{attribute 'linkalways'} 
{attribute 'no_explicit_call' := 'This FB is a CLASS and must be accessed using methods or properties'}
{attribute 'enable_dynamic_creation'}
FUNCTION_BLOCK Node_F_VN_ElementwiseLog EXTENDS VisionNode
VAR
    ipSrcImage : _ITcVnImage;
    ipDestImage : _ITcVnImage;
    hrPrev : _HRESULT(S_OK);
	hresult : _HRESULT(S_OK);
END_VAR

METHOD PUBLIC  Clone : I_Node
VAR
	pNode : POINTER TO Node_F_VN_ElementwiseLog;
END_VAR
pNode := __NEW(Node_F_VN_ElementwiseLog);
Clone := pNode^;
END_METHOD

METHOD FB_init : BOOL
VAR_INPUT
	bInitRetains : BOOL; // if TRUE, the retain variables are initialized (warm start / cold start)
	bInCopyCode : BOOL;  // if TRUE, the instance afterwards gets moved into the copy code (online change)
END_VAR
AddInput('ipSrcImage', ipSrcImage);
AddInput('hrPrev', hrPrev);
AddOutput('ipDestImage', ipDestImage);
AddOutput('hresult',hresult);
END_METHOD

METHOD PROTECTED OnExecute : HRESULT
hresult.Value := F_VN_ElementwiseLog(
    ipSrcImage := ipSrcImage.Value,
	ipDestImage := ipDestImage.Value,
	hrPrev:= hrPrev.Value);
END_METHOD

METHOD PUBLIC PreExecutionCheck
VAR_INPUT
	Check : I_PreExecutionChecks;
END_VAR
IF FAILED(hrPrev.Value) THEN
    RETURN;
END_IF

Check.IsTrue(ipSrcImage.IsValid, 'ipSrcImage must contain an image');
Check.IsTrue((ipSrcImage.IsPixelDepth(32) OR
              ipSrcImage.IsPixelDepth(64)), 'ipSrcImage must have 32 or 64 bit pixel depth');
END_METHOD

END_FUNCTION_BLOCK

(* stored: Version 1.1.0.1, ProductVersion 3.1.4024.13
   POU Node_F_VN_ElementwiseLog: Id {b1fc8eca-c2ac-0d25-192a-01f05aab5338}, SpecialFunc None
   Folder Constructor: Id {22ff3e3f-64d5-0cb8-344a-76288229d708}
   Method Clone: Id {07300f5c-d289-0387-08dd-af41adda509a}
   Method FB_init: Id {4a9236fe-a0ec-0926-278e-4d2b32131453}
   Method OnExecute: Id {be71dc6b-172b-0212-1a3b-923bedb3957a}
   Method PreExecutionCheck: Id {990add5a-c363-02fa-2d54-cb2138782aeb} *)
